TYPE LEDColor :
STRUCT	
	red 	:USINT;
	green	:USINT;
	blue	:USINT;
	white	:USINT;
END_STRUCT
END_TYPE

(* stored: Version 1.1.0.1, ProductVersion 3.1.4026.18
   DUT LEDColor: Id {7a84a1ca-42c1-49cd-81ce-655267b307c3} *)
